(* IEC 61131-3 sources: ot-sentinel-lite/artifacts/icspector/incident, 1 file *)

(* ---- conveyor_logic.st ---- *)
VAR
  Jam_Timeout : TIME := T#20s;
END_VAR
